FUNCTION_BLOCK HCylAdpOL (* Composite Function Block Type *)
  (* Standard: 61499-2 *)
  (* Version 0.0, 06/10/2018, Atmojo, nxtControl GmbH, template *)
  PACKAGE Main;
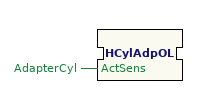
  SOCKETS
    ActSens : AdapterCyl;
  END_SOCKETS
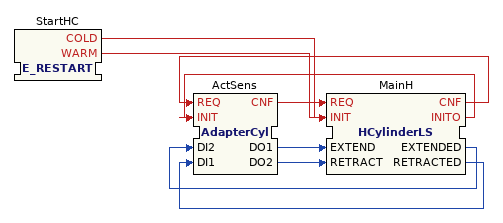
  FBS
    MainH : HCylinderLS;
    StartHC : E_RESTART;
  END_FBS
  EVENT_CONNECTIONS
    ActSens.CNF TO MainH.REQ;
    StartHC.COLD TO MainH.INIT;
    StartHC.WARM TO MainH.INIT;
    MainH.CNF TO ActSens.REQ;
    MainH.INITO TO ActSens.INIT;
  END_CONNECTIONS
  DATA_CONNECTIONS
    ActSens.DO1 TO MainH.EXTEND;
    ActSens.DO2 TO MainH.RETRACT;
    MainH.EXTENDED TO ActSens.DI2;
    MainH.RETRACTED TO ActSens.DI1;
  END_CONNECTIONS
END_FUNCTION_BLOCK
